FUNCTION_BLOCK ROBOT5TESTFB (* JADE WORKER *)
  (* Standard: 61499-1 *)
  (* Version 1.0, 2014-04-22, Ahmed, Fraunhofer IGD *)
  (* Compiler header: package fb.rt; *)
  (* Compiler Java Sun JDK 1.5.0 *)
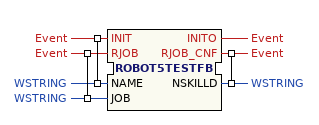
  EVENT_INPUT
    INIT WITH NAME; (* Normal Execution Request *)
    RJOB WITH JOB; (* Normal Execution Request *)
  END_EVENT
  EVENT_OUTPUT
    INITO; (* Execution Confirmation *)
    RJOB_CNF WITH NSKILLD; (* Execution Confirmation *)
  END_EVENT
  VAR_INPUT
    NAME : WSTRING;
    JOB : WSTRING;
  END_VAR
  VAR_OUTPUT
    NSKILLD : WSTRING;
  END_VAR
END_FUNCTION_BLOCK
